// TwinCAT 3 PLC project StructureText_ex
// ProgramVersion: 3.1.4023.0
// libraries:
//   Tc2_Standard, * (Beckhoff Automation GmbH)
//   Tc2_System, * (Beckhoff Automation GmbH)
//   Tc3_Module, * (Beckhoff Automation GmbH)
// project tree:
//   / PlcTask.TcTTO
//   POUs/ MAIN.TcPOU, struct_text_ex.TcPOU
// real-time tasks:
//   TASK PlcTask: cycle T#10ms, priority 20, ADS port 350

CONFIGURATION StructureText_ex
    RESOURCE PLC ON TwinCAT3
        TASK PlcTask(INTERVAL := T#10ms, PRIORITY := 20);
        PROGRAM MAIN WITH PlcTask : MAIN;
    END_RESOURCE
END_CONFIGURATION

// ---- POUs/MAIN.TcPOU
PROGRAM MAIN
VAR
END_VAR

struct_text_ex();

END_PROGRAM

// ---- POUs/struct_text_ex.TcPOU
PROGRAM struct_text_ex
VAR
	Buttons: ARRAY [1..2] OF BOOL;
	Coils: ARRAY[1..5] OF BOOL;
	OverCurrent: ARRAY[1..5] OF BOOL;
	valves: ARRAY[1..5] OF BOOL;
	Ultrasonic: INT:=800;
	Threshold: INT :=200;
	index:INT;
	
END_VAR

IF Buttons[1] = TRUE AND Buttons[2] = FALSE THEN
	FOR index:=1 TO 4 BY 1 DO
		IF OverCurrent[index] OR Valves[index]=FALSE THEN
			Coils[index]:=FALSE;
		ELSE
			IF Ultrasonic >= Threshold THEN
				Coils[index]:=TRUE;
			ELSE
				Coils[index]:=FALSE;
			END_IF
		END_IF
	END_FOR
END_IF

IF Buttons[1] = TRUE AND Buttons[2] = FALSE THEN
	IF OverCurrent[5] OR Valves[5]=FALSE THEN
		Coils[5]:=TRUE;
	ELSE
		IF Ultrasonic < Threshold THEN
			Coils[5]:= TRUE;
		END_IF
	END_IF
END_IF

END_PROGRAM
